FUNCTION_BLOCK INTERNAL FB_ActivateAction EXTENDS FB_Action
VAR
    _bActivated: BOOL;
END_VAR

METHOD  Execute
VAR_INPUT
    ipObject: I_Object;
END_VAR
VAR
    p: POINTER TO FB_ActionTestObject;
END_VAR
__QUERYPOINTER(ipObject, p);

IF p <> 0 THEN
    p^.Activate(THIS^._bActivated);
END_IF
END_METHOD

METHOD Inputs : I_Action
VAR_INPUT
    bActivate: BOOL;
END_VAR
Inputs := THIS^;
THIS^._bActivated := bActivate;
END_METHOD

END_FUNCTION_BLOCK

(* stored: Version 1.1.0.1, ProductVersion 3.1.4024.12
   POU FB_ActivateAction: Id {2b7d7fab-da5a-0021-1eae-a8188ca21e2e}, SpecialFunc None
   Method Execute: Id {a913cb0f-008f-0ba3-36a1-85b87f9eb84c}
   Method Inputs: Id {b381ba14-5d21-07eb-211b-2bb001f3cf73} *)
